FUNCTION_BLOCK IP_CONTROL_RESET
VAR_INPUT
END_VAR
VAR_OUTPUT
	READY : BOOL;
END_VAR
VAR
	fbSocketCloseAll : FB_SocketCloseAll;
	step : BYTE;
END_VAR

(* On PLC reset or program download close all old connections *)

CASE TCP_SERVER_RESET OF

2:	READY := TRUE;
	RETURN;

1:	IF step = 0 THEN
		RETURN;
	END_IF;

0:	TCP_SERVER_RESET := 1; (* Reset ist aktiv *)
	step := 1;

END_CASE;

CASE step OF

0:	RETURN;

1:	fbSocketCloseAll(sSrvNetId:= '', bExecute:= TRUE, tTimeout:= T#10s );
	step := 2;

2:	fbSocketCloseAll(bExecute:= FALSE);
	IF fbSocketCloseAll.bBusy = FALSE THEN
		step := 0;
		TCP_SERVER_RESET := 2; (* Reset durchgeführt , Bereit zur Verwendung *)
	END_IF;

END_CASE;

END_FUNCTION_BLOCK

(* stored: Version 1.1.0.1, ProductVersion 3.1.4024.9
   POU IP_CONTROL_RESET: Id {9000eaca-c207-49aa-bb20-d9fd11ce797f}, SpecialFunc None *)
